{attribute 'qualified_only'}
{attribute 'strict'}
TYPE  E_WashProgram :
(
	NONE      := 0,
    ECO       := 1,
    NORMAL    := 2,
    INTENSIVE := 3
);
END_TYPE

(* stored: Version 1.1.0.1, ProductVersion 3.1.4024.16
   DUT E_WashProgram: Id {7f529343-3922-4ec6-99c1-5a7ab6c42cb8} *)
